{attribute 'linkalways'} 
{attribute 'no_explicit_call' := 'This FB is a CLASS and must be accessed using methods or properties'}
{attribute 'enable_dynamic_creation'}
FUNCTION_BLOCK _Array0to9OfITcVnImage EXTENDS ArrayDatatypeBase_1D
VAR CONSTANT
	lBound : DINT := 0;
	uBound : DINT := 9;
END_VAR
VAR
	localData : ARRAY [lBound..uBound] OF ITcVnImage;
	activeData : REFERENCE TO ARRAY [lBound..uBound] OF ITcVnImage REF= localData;
	elements : ARRAY [lBound..uBound] OF _ITcVnImage;
	baseType : _ITcVnImage;
END_VAR

PROPERTY PUBLIC Address : PVOID
GET
Address := ADR(activeData);
END_GET
END_PROPERTY

PROPERTY PUBLIC BaseDatatype : I_Datatype
GET
BaseDatatype := baseType;
END_GET
END_PROPERTY

METHOD PUBLIC ClearReference
VAR_INPUT
END_VAR
activeData REF= localData;
SetElementReference();
END_METHOD

METHOD PUBLIC Clone : I_Datatype
VAR
    pClone : POINTER TO _Array0to9OfITcVnImage;
END_VAR
pClone := __NEW(_Array0to9OfITcVnImage());
pClone^.Value := Value;
Clone := pClone^;
END_METHOD

METHOD FB_init : BOOL
VAR_INPUT
	bInitRetains : BOOL; // if TRUE, the retain variables are initialized (warm start / cold start)
	bInCopyCode : BOOL;  // if TRUE, the instance afterwards gets moved into the copy code (online change)
END_VAR
SetElementReference();
END_METHOD

METHOD PUBLIC MakeReferenceTo
VAR_INPUT
	ReferenceTarget : REFERENCE TO ARRAY [lBound..uBound] OF ITcVnImage;
END_VAR
activeData REF= ReferenceTarget;
SetElementReference();
END_METHOD

METHOD PROTECTED OnSerializeArrayValues
VAR_INPUT
	Serializer : I_Serializer;
END_VAR
VAR
	i : DINT;
END_VAR
FOR i := lBound TO uBound DO
	elements[i].SerializeWith(Serializer);
END_FOR
END_METHOD

METHOD PROTECTED SetElementReference
VAR_INPUT
END_VAR
VAR
	i : DINT;
END_VAR
FOR i := lBound TO uBound DO
	elements[i].MakeReferenceTo(activeData[i]);
END_FOR
END_METHOD

PROPERTY PUBLIC Size : UDINT
GET
Size := SIZEOF(activeData);
END_GET
END_PROPERTY

METHOD PROTECTED TryDeserializeArrayValues : BOOL
VAR_INPUT
	Deserializer : I_Deserializer;
	Feedback : I_DeserializerFeedback;
END_VAR
VAR
	enumerator : I_DeserializerArrayForwardEnumerator;
	i : DINT;
END_VAR
enumerator := Deserializer.GetArrayEnumerator();
i := lBound;

WHILE enumerator.MoveNext() AND i <= uBound DO
	
	IF NOT elements[i].TryDeserializeFrom(enumerator.Current, Feedback) THEN
		EXIT;
	END_IF
	i := i + 1;

END_WHILE
enumerator.Dispose();
END_METHOD

METHOD PUBLIC TryGetElementAsDatatypeByIndex : BOOL
VAR_INPUT
	Index : DINT;
	Destination : REFERENCE TO I_Datatype;
END_VAR
IF Index < lbound OR Index > ubound THEN
	RETURN;
END_IF

Destination := elements[Index];
TryGetElementAsDatatypeByIndex := TRUE;
END_METHOD

METHOD PUBLIC TryGetLowerBound : BOOL
VAR_INPUT
	Dimention : UDINT;
	Destination : REFERENCE TO DINT;
END_VAR
IF Dimention = 1 THEN
	Destination := lBound;
	TryGetLowerBound := TRUE;
END_IF
END_METHOD

METHOD PUBLIC TryGetUpperBound : BOOL
VAR_INPUT
	Dimention : UDINT;
	Destination : REFERENCE TO DINT;
END_VAR
IF Dimention = 1 THEN
	Destination := uBound;
	TryGetUpperBound := TRUE;
END_IF
END_METHOD

METHOD TryMakeReferenceTo : BOOL
VAR_INPUT
	Target : I_Datatype;
END_VAR
VAR
	pTargetData : POINTER TO ARRAY [lBound..uBound] OF ITcVnImage;
END_VAR
IF NOT IsEquivalentTo(Target) THEN
	RETURN;
END_IF

pTargetData := Target.Address;
activeData REF= pTargetData^;
SetElementReference();
TryMakeReferenceTo := TRUE;
END_METHOD

PROPERTY PUBLIC Value : REFERENCE TO ARRAY [lBound..uBound] OF ITcVnImage;
GET
Value ref= activeData;
END_GET
END_PROPERTY

END_FUNCTION_BLOCK

(* stored: Version 1.1.0.1, ProductVersion 3.1.4024.13
   POU _Array0to9OfITcVnImage: Id {53378396-ddd0-01d6-1fe9-e5bade8d0852}, SpecialFunc None
   Folder Core: Id {cf0b6631-3d92-077e-1e52-81dfeb713bea}
   Folder Constructor: Id {7e5a5611-d143-024e-1c43-1b4eaee33bfb}
   Folder Protected: Id {6b0f9b82-5c01-00a2-1a1c-bc3043fa0735}
   Folder Customize: Id {6082933d-8e3c-03d6-17ac-83eed2eb385f}
   Property Address: Id {c9537324-d83d-07f2-2427-55ad2947f976}
   Get Get: Id {540c7a6c-50c2-0678-3632-b18b09bcc947}
   Property BaseDatatype: Id {dcfeb457-216c-0f4d-1cb0-1a67dc03fc55}
   Get Get: Id {cd6b0f17-65eb-0ec4-3a35-e381886a164a}
   Method ClearReference: Id {bb83f288-35cd-0262-1403-ae7f8482d876}
   Method Clone: Id {a45e0e84-1483-0d52-2184-26fe9c42b26e}
   Method FB_init: Id {a65fec8e-7cfb-0c62-0176-fb0c82dd4ae7}
   Method MakeReferenceTo: Id {679eb237-e4c1-0b1d-271a-f2529878e181}
   Method OnSerializeArrayValues: Id {bf75be3b-9faf-05fe-1164-ae9d6cf29977}
   Method SetElementReference: Id {ff638f2e-9245-0b2a-0a25-3c72ece7fa3c}
   Property Size: Id {233853ae-e1f6-08ba-1d68-0844b8240150}
   Get Get: Id {73ce24e9-f83a-0c96-09d3-d48ae650e93c}
   Method TryDeserializeArrayValues: Id {2e44b3ef-9532-0147-1ae6-3869d7e8c373}
   Method TryGetElementAsDatatypeByIndex: Id {0086506a-a05e-0bc0-2ea4-53467d5fe235}
   Method TryGetLowerBound: Id {80329649-e17c-04fe-3774-d39ddf7c135a}
   Method TryGetUpperBound: Id {77537e3a-48fa-00d1-2ae0-45c3c2591ea5}
   Method TryMakeReferenceTo: Id {e540e74c-b883-0bc0-2019-6dd7114ce613}
   Property Value: Id {96672d1c-be7f-0582-2f79-66e8b61430a4}
   Get Get: Id {68fe547c-9461-01fe-01f1-6ee341c80324} *)
